Staubli VAL3: launch_print.pgx

program launch_print()
begin

  // ouverture obturateur
    dioSet(doValve1,0)
    dioSet(doValve2,1)
    put("Obturateur ouvert")
    delay(2)
    // mise en marche pompe vitesse faible
    dioSet(doPompe,1)
    put("Pompe en marche")
    // mise en rotation pompe vitesse donnée
    aioSet(Tpompe,0.2)
    put("Pompe en rotation")
    delay(1)

end
